PROGRAM ReadMe

(*

Function Block
 - InOutput, InPut, Output are intended to use from other program
 - Properties are intended for Encapsulation
































*)

END_PROGRAM

(* stored: Version 1.1.0.1, ProductVersion 3.1.4024.12
   POU ReadMe: Id {11cc9a99-5513-415e-98e2-65b91c9f23a1}, SpecialFunc None *)
